Universal Robots PolyScope program: ret.urp

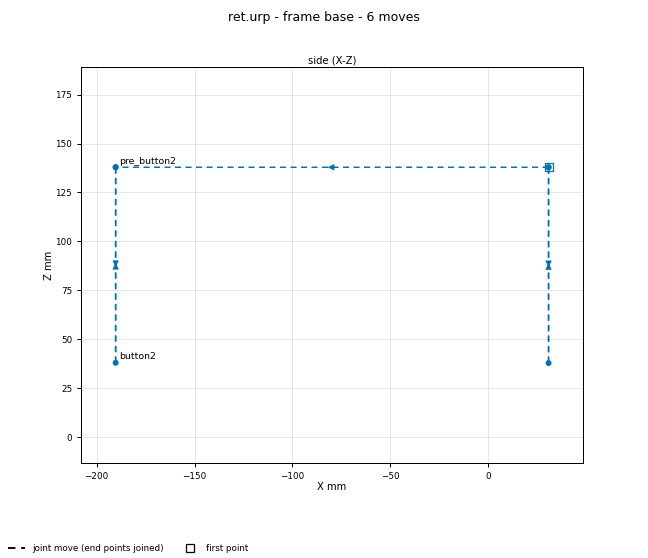
[picture p0: tool path of ret.urp in frame base, 6 of 6 moves have a stored position in this frame; points joined in program order, loops and branches not executed]
Program ret (installation=default directory=/programs/usbdisk/programs createdIn=5.2.1.61344 lastSavedIn=5.2.1.61344 robotSerialNumber=20185500910)
Calibrated DH parameters: a=[0.000049, -0.2988, -0.136614, -0.000051, 0.000155, 0]; d=[0.162579, 88.949821, -241.716128, 152.899954, 0.099639, 0.099482]; alpha=[1.56987, -0.003405, -0.002407, 1.569674, -1.569166, 0]; deltaTheta=[0, -0.792152, 8.290367, -1.215029, 0.000002, 0]
BeforeStart
  var_1 := socket_open("192.168.56.1",65432)
Robot Program (runOnlyOnce=false)
  Loop While (checkContinuously=false) expression=(var_1≟ False )
    var_1 := socket_open("192.168.56.1",65432)
    Wait Sleep waitTime=0.5
  MoveJ speed 60 deg/s, acceleration 80 deg/s^2 (useActiveTCP=true) feature=Base
    Waypoint pre_button1: TCP in base x=30.846 y=-395.628 z=137.884 mm, rx=-0.0044 ry=3.138 rz=-0.0014 rad; joints [-66.21, -82.351, -130.278, -57.335, 89.99, 23.802] deg; TCP offset x=0 y=0 z=135 mm, rx=0 ry=0 rz=0 rad
  MoveJ speed 60 deg/s, acceleration 80 deg/s^2 (useActiveTCP=true) feature=Base
    Waypoint button1: TCP in base x=30.847 y=-395.635 z=37.874 mm, rx=-0.0044 ry=3.138 rz=-0.0014 rad; joints [-66.177, -95.129, -137.923, -36.913, 89.937, 23.763] deg; TCP offset x=0 y=0 z=135 mm, rx=0 ry=0 rz=0 rad
  Script: socket_send_string("ur_native;time;1")
  MoveJ speed 60 deg/s, acceleration 80 deg/s^2 (useActiveTCP=true) feature=Base
    Waypoint post_button1: TCP in base x=30.834 y=-395.635 z=137.895 mm, rx=-0.0044 ry=3.138 rz=-0.0014 rad; joints [-66.211, -82.351, -130.276, -57.337, 89.988, 23.801] deg; TCP offset x=0 y=0 z=135 mm, rx=0 ry=0 rz=0 rad
  MoveJ speed 60 deg/s, acceleration 80 deg/s^2 (useActiveTCP=true) feature=Base
    Waypoint pre_button2: TCP in base x=-190.305 y=-395.726 z=137.88 mm, rx=-0.0043 ry=3.138 rz=-0.0013 rad; joints [-98.293, -88.745, -124.486, -56.843, 90.016, -8.293] deg; TCP offset x=0 y=0 z=135 mm, rx=0 ry=0 rz=0 rad
  MoveJ speed 60 deg/s, acceleration 80 deg/s^2 (useActiveTCP=true) feature=Base
    Waypoint button2: TCP in base x=-190.322 y=-395.731 z=37.997 mm, rx=-0.0043 ry=3.138 rz=-0.0015 rad; joints [-98.269, -100.289, -131.454, -38.324, 89.97, -8.336] deg; TCP offset x=0 y=0 z=135 mm, rx=0 ry=0 rz=0 rad
  Script: socket_send_string("ur_native;time;2")
  MoveJ speed 60 deg/s, acceleration 80 deg/s^2 (useActiveTCP=true) feature=Base
    Waypoint post_button2: TCP in base x=-190.314 y=-395.727 z=137.988 mm, rx=-0.0042 ry=3.138 rz=-0.0015 rad; joints [-98.294, -88.734, -124.479, -56.856, 90.015, -8.29] deg
  var_1 := False
  Script: socket_close()
